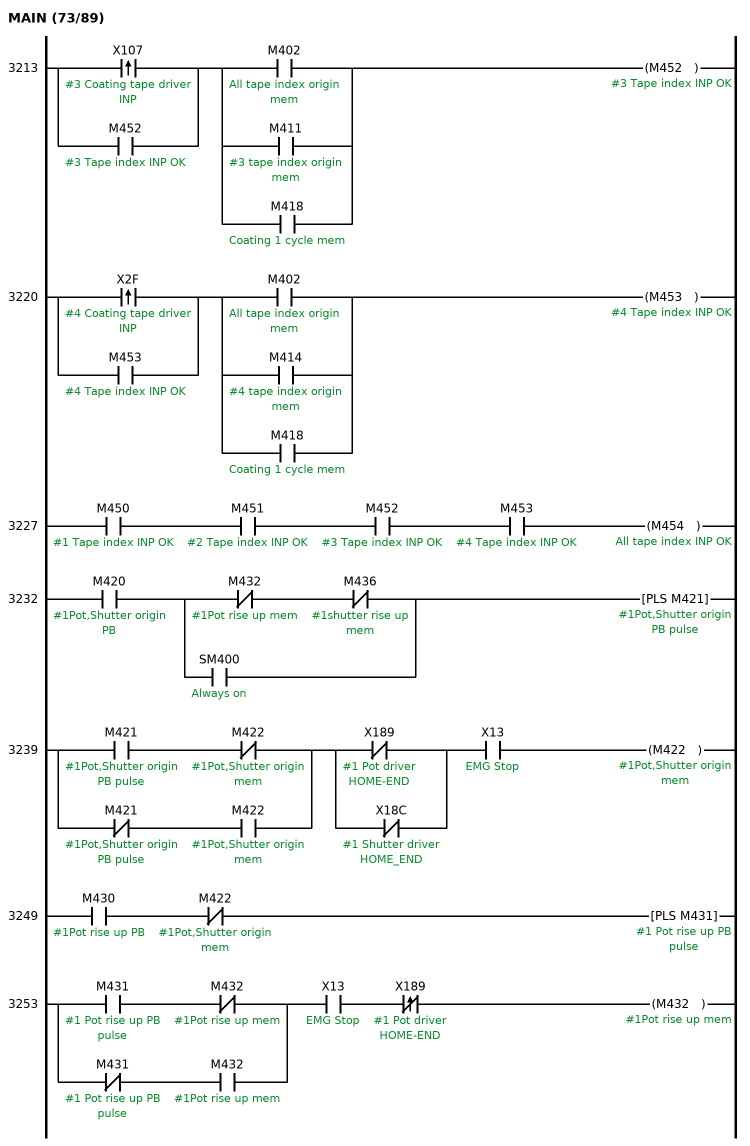
[picture p72: ladder of MAIN, rungs at steps 3213 to 3253]
3213  LDP     X107  ; #3 Coating tape driver INP
      OR      M452  ; #3 Tape index INP OK
      LD      M402  ; All tape index origin mem
      OR      M411  ; #3 tape index origin mem
      OR      M418  ; Coating 1 cycle mem
      ANB
      OUT     M452  ; #3 Tape index INP OK
3220  LDP     X2F  ; #4 Coating tape driver INP
      OR      M453  ; #4 Tape index INP OK
      LD      M402  ; All tape index origin mem
      OR      M414  ; #4 tape index origin mem
      OR      M418  ; Coating 1 cycle mem
      ANB
      OUT     M453  ; #4 Tape index INP OK
3227  LD      M450  ; #1 Tape index INP OK
      AND     M451  ; #2 Tape index INP OK
      AND     M452  ; #3 Tape index INP OK
      AND     M453  ; #4 Tape index INP OK
      OUT     M454  ; All tape index INP OK
3232  LD      M420  ; #1Pot,Shutter origin PB
      LDI     M432  ; #1Pot rise up mem
      ANI     M436  ; #1shutter rise up mem
      OR      SM400  ; Always on
      ANB
      PLS     M421  ; #1Pot,Shutter origin PB pulse
3239  LD      M421  ; #1Pot,Shutter origin PB pulse
      ANI     M422  ; #1Pot,Shutter origin mem
      LDI     M421  ; #1Pot,Shutter origin PB pulse
      AND     M422  ; #1Pot,Shutter origin mem
      ORB
      LDI     X189  ; #1 Pot driver HOME-END
      ORI     X18C  ; #1 Shutter driver HOME_END
      ANB
      AND     X13  ; EMG Stop
      OUT     M422  ; #1Pot,Shutter origin mem
3249  LD      M430  ; #1Pot rise up PB
      ANI     M422  ; #1Pot,Shutter origin mem
      PLS     M431  ; #1 Pot rise up PB pulse
3253  LD      M431  ; #1 Pot rise up PB pulse
      ANI     M432  ; #1Pot rise up mem
      LDI     M431  ; #1 Pot rise up PB pulse
      AND     M432  ; #1Pot rise up mem
      ORB
      AND     X13  ; EMG Stop
      ANDPI   X189  ; #1 Pot driver HOME-END
      OUT     M432  ; #1Pot rise up mem
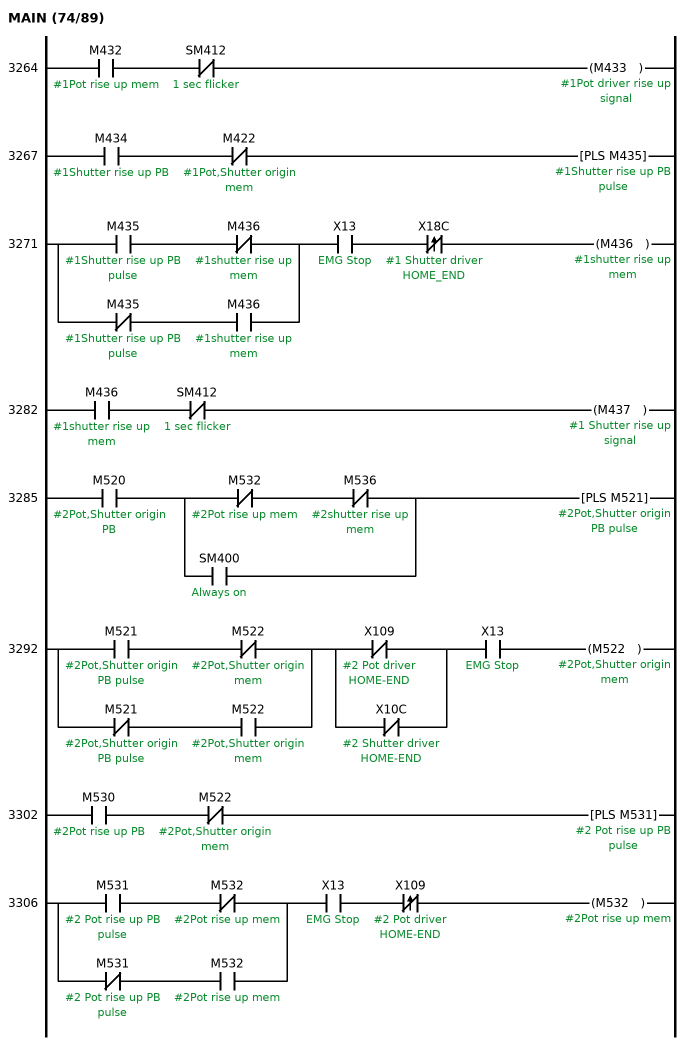
3264  LD      M432  ; #1Pot rise up mem
      ANI     SM412  ; 1 sec flicker
      OUT     M433  ; #1Pot driver rise up signal
3267  LD      M434  ; #1Shutter rise up PB
      ANI     M422  ; #1Pot,Shutter origin mem
      PLS     M435  ; #1Shutter rise up PB pulse
3271  LD      M435  ; #1Shutter rise up PB pulse
      ANI     M436  ; #1shutter rise up mem
      LDI     M435  ; #1Shutter rise up PB pulse
      AND     M436  ; #1shutter rise up mem
      ORB
      AND     X13  ; EMG Stop
      ANDPI   X18C  ; #1 Shutter driver HOME_END
      OUT     M436  ; #1shutter rise up mem
3282  LD      M436  ; #1shutter rise up mem
      ANI     SM412  ; 1 sec flicker
      OUT     M437  ; #1 Shutter rise up signal
3285  LD      M520  ; #2Pot,Shutter origin PB
      LDI     M532  ; #2Pot rise up mem
      ANI     M536  ; #2shutter rise up mem
      OR      SM400  ; Always on
      ANB
      PLS     M521  ; #2Pot,Shutter origin PB pulse
3292  LD      M521  ; #2Pot,Shutter origin PB pulse
      ANI     M522  ; #2Pot,Shutter origin mem
      LDI     M521  ; #2Pot,Shutter origin PB pulse
      AND     M522  ; #2Pot,Shutter origin mem
      ORB
      LDI     X109  ; #2 Pot driver HOME-END
      ORI     X10C  ; #2 Shutter driver HOME-END
      ANB
      AND     X13  ; EMG Stop
      OUT     M522  ; #2Pot,Shutter origin mem
3302  LD      M530  ; #2Pot rise up PB
      ANI     M522  ; #2Pot,Shutter origin mem
      PLS     M531  ; #2 Pot rise up PB pulse
3306  LD      M531  ; #2 Pot rise up PB pulse
      ANI     M532  ; #2Pot rise up mem
      LDI     M531  ; #2 Pot rise up PB pulse
      AND     M532  ; #2Pot rise up mem
      ORB
      AND     X13  ; EMG Stop
      ANDPI   X109  ; #2 Pot driver HOME-END
      OUT     M532  ; #2Pot rise up mem
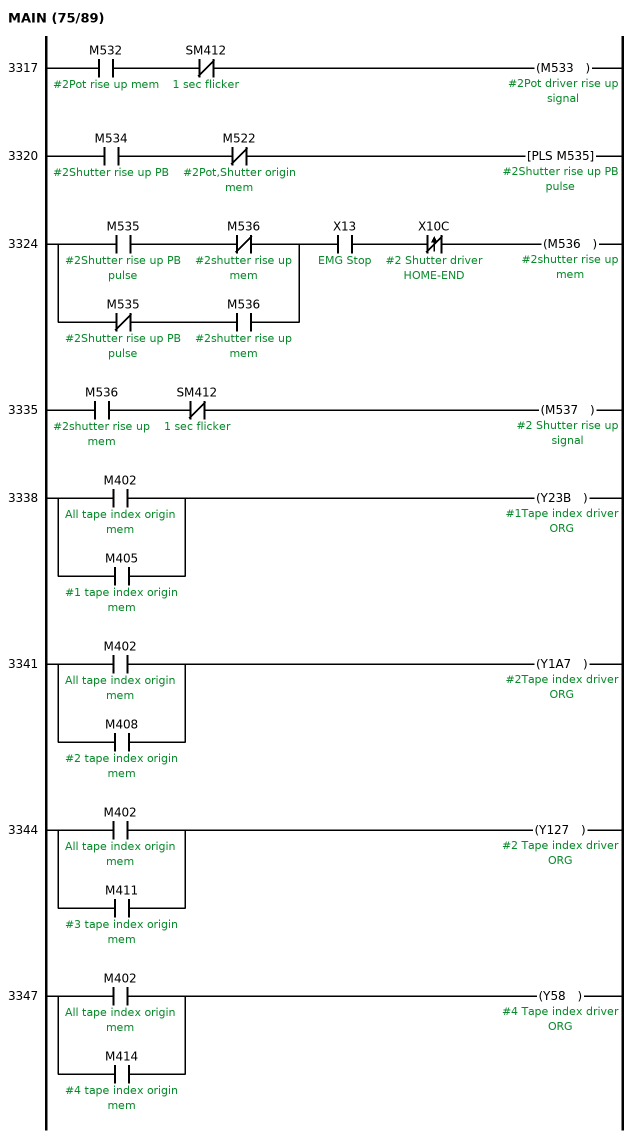
3317  LD      M532  ; #2Pot rise up mem
      ANI     SM412  ; 1 sec flicker
      OUT     M533  ; #2Pot driver rise up signal
3320  LD      M534  ; #2Shutter rise up PB
      ANI     M522  ; #2Pot,Shutter origin mem
      PLS     M535  ; #2Shutter rise up PB pulse
3324  LD      M535  ; #2Shutter rise up PB pulse
      ANI     M536  ; #2shutter rise up mem
      LDI     M535  ; #2Shutter rise up PB pulse
      AND     M536  ; #2shutter rise up mem
      ORB
      AND     X13  ; EMG Stop
      ANDPI   X10C  ; #2 Shutter driver HOME-END
      OUT     M536  ; #2shutter rise up mem
3335  LD      M536  ; #2shutter rise up mem
      ANI     SM412  ; 1 sec flicker
      OUT     M537  ; #2 Shutter rise up signal
3338  LD      M402  ; All tape index origin mem
      OR      M405  ; #1 tape index origin mem
      OUT     Y23B  ; #1Tape index driver ORG
3341  LD      M402  ; All tape index origin mem
      OR      M408  ; #2 tape index origin mem
      OUT     Y1A7  ; #2Tape index driver ORG
3344  LD      M402  ; All tape index origin mem
      OR      M411  ; #3 tape index origin mem
      OUT     Y127  ; #2 Tape index driver ORG
3347  LD      M402  ; All tape index origin mem
      OR      M414  ; #4 tape index origin mem
      OUT     Y58  ; #4 Tape index driver ORG
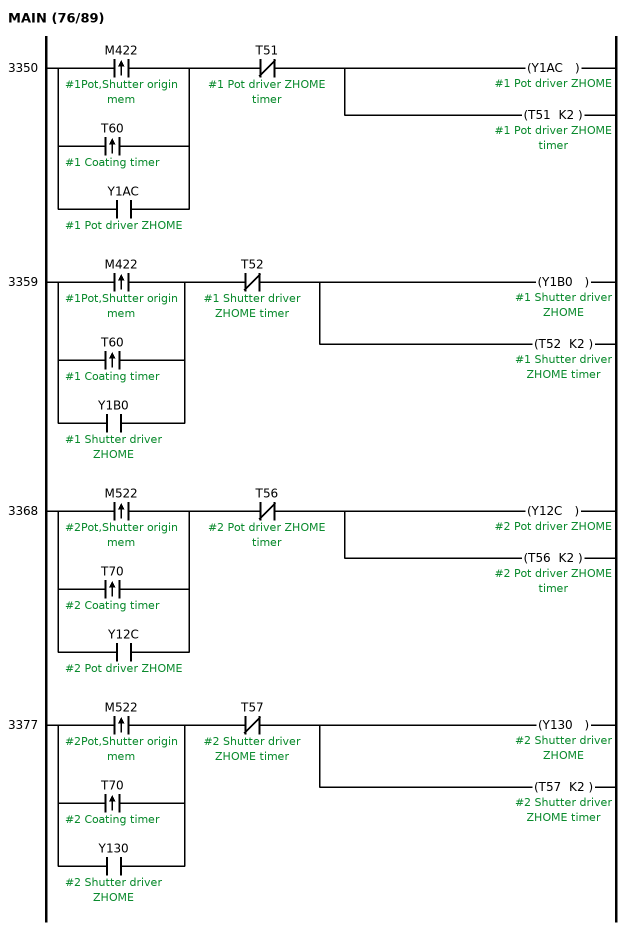
3350  LDP     M422  ; #1Pot,Shutter origin mem
      ORP     T60  ; #1 Coating timer
      OR      Y1AC  ; #1 Pot driver ZHOME
      ANI     T51  ; #1 Pot driver ZHOME timer
      OUT     Y1AC  ; #1 Pot driver ZHOME
      OUT     T51 K2  ; #1 Pot driver ZHOME timer
3359  LDP     M422  ; #1Pot,Shutter origin mem
      ORP     T60  ; #1 Coating timer
      OR      Y1B0  ; #1 Shutter driver ZHOME
      ANI     T52  ; #1 Shutter driver ZHOME timer
      OUT     Y1B0  ; #1 Shutter driver ZHOME
      OUT     T52 K2  ; #1 Shutter driver ZHOME timer
3368  LDP     M522  ; #2Pot,Shutter origin mem
      ORP     T70  ; #2 Coating timer
      OR      Y12C  ; #2 Pot driver ZHOME
      ANI     T56  ; #2 Pot driver ZHOME timer
      OUT     Y12C  ; #2 Pot driver ZHOME
      OUT     T56 K2  ; #2 Pot driver ZHOME timer
3377  LDP     M522  ; #2Pot,Shutter origin mem
      ORP     T70  ; #2 Coating timer
      OR      Y130  ; #2 Shutter driver ZHOME
      ANI     T57  ; #2 Shutter driver ZHOME timer
      OUT     Y130  ; #2 Shutter driver ZHOME
      OUT     T57 K2  ; #2 Shutter driver ZHOME timer
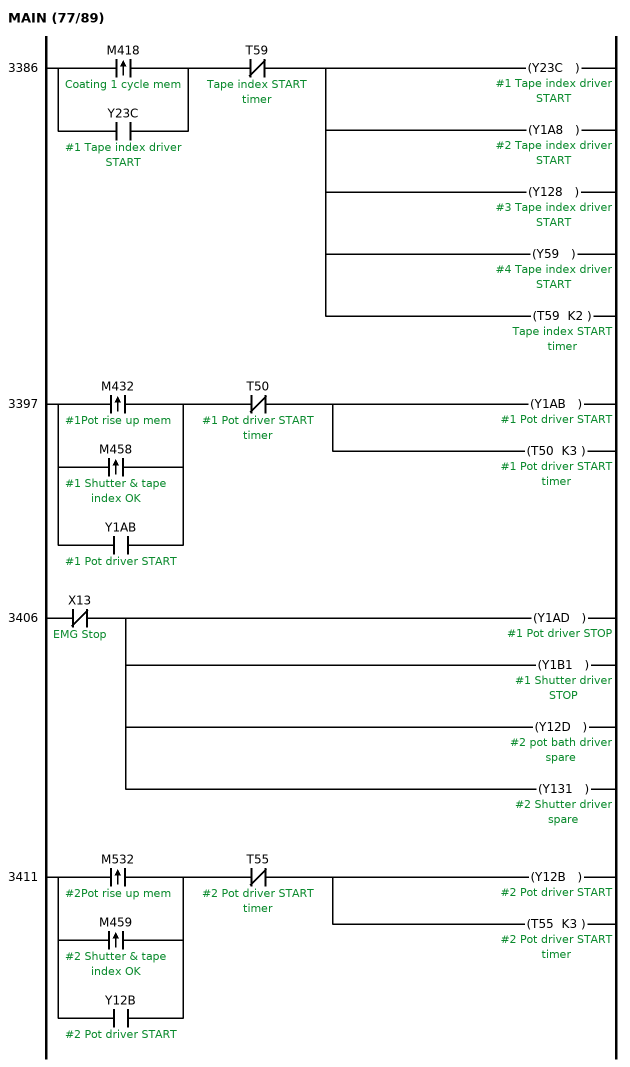
3386  LDP     M418  ; Coating 1 cycle mem
      OR      Y23C  ; #1 Tape index driver START
      ANI     T59  ; Tape index START timer
      OUT     Y23C  ; #1 Tape index driver START
      OUT     Y1A8  ; #2 Tape index driver START
      OUT     Y128  ; #3 Tape index driver START
      OUT     Y59  ; #4 Tape index driver START
      OUT     T59 K2  ; Tape index START timer
3397  LDP     M432  ; #1Pot rise up mem
      ORP     M458  ; #1 Shutter & tape index OK
      OR      Y1AB  ; #1 Pot driver START
      ANI     T50  ; #1 Pot driver START timer
      OUT     Y1AB  ; #1 Pot driver START
      OUT     T50 K3  ; #1 Pot driver START timer
3406  LDI     X13  ; EMG Stop
      OUT     Y1AD  ; #1 Pot driver STOP
      OUT     Y1B1  ; #1 Shutter driver STOP
      OUT     Y12D  ; #2 pot bath driver spare
      OUT     Y131  ; #2 Shutter driver spare
3411  LDP     M532  ; #2Pot rise up mem
      ORP     M459  ; #2 Shutter & tape index OK
      OR      Y12B  ; #2 Pot driver START
      ANI     T55  ; #2 Pot driver START timer
      OUT     Y12B  ; #2 Pot driver START
      OUT     T55 K3  ; #2 Pot driver START timer
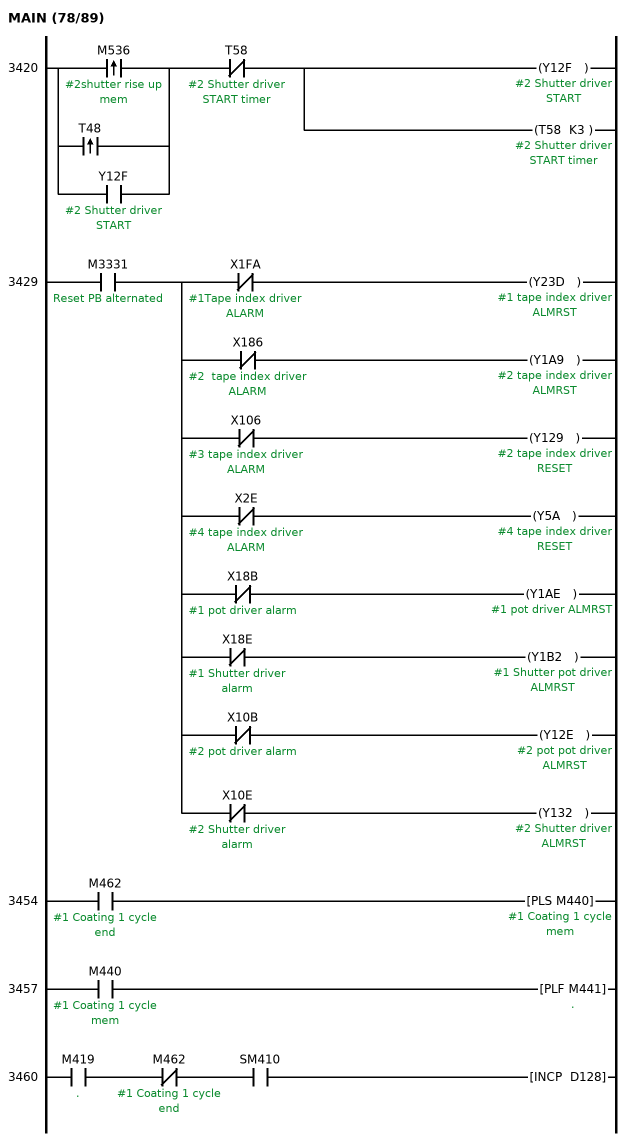
3420  LDP     M536  ; #2shutter rise up mem
      ORP     T48
      OR      Y12F  ; #2 Shutter driver START
      ANI     T58  ; #2 Shutter driver START timer
      OUT     Y12F  ; #2 Shutter driver START
      OUT     T58 K3  ; #2 Shutter driver START timer
3429  LD      M3331  ; Reset PB alternated
      MPS
      ANI     X1FA  ; #1Tape index driver ALARM
      OUT     Y23D  ; #1 tape index driver ALMRST
      MRD
      ANI     X186  ; #2  tape index driver ALARM
      OUT     Y1A9  ; #2 tape index driver ALMRST
      MRD
      ANI     X106  ; #3 tape index driver ALARM
      OUT     Y129  ; #2 tape index driver RESET
      MRD
      ANI     X2E  ; #4 tape index driver ALARM
      OUT     Y5A  ; #4 tape index driver RESET
      MRD
      ANI     X18B  ; #1 pot driver alarm
      OUT     Y1AE  ; #1 pot driver ALMRST
      MRD
      ANI     X18E  ; #1 Shutter driver alarm
      OUT     Y1B2  ; #1 Shutter pot driver ALMRST
      MRD
      ANI     X10B  ; #2 pot driver alarm
      OUT     Y12E  ; #2 pot pot driver ALMRST
      MPP
      ANI     X10E  ; #2 Shutter driver alarm
      OUT     Y132  ; #2 Shutter driver ALMRST
3454  LD      M462  ; #1 Coating 1 cycle end
      PLS     M440  ; #1 Coating 1 cycle mem
3457  LD      M440  ; #1 Coating 1 cycle mem
      PLF     M441  ; .
3460  LD      M419  ; .
      ANI     M462  ; #1 Coating 1 cycle end
      AND     SM410
      INCP    D128
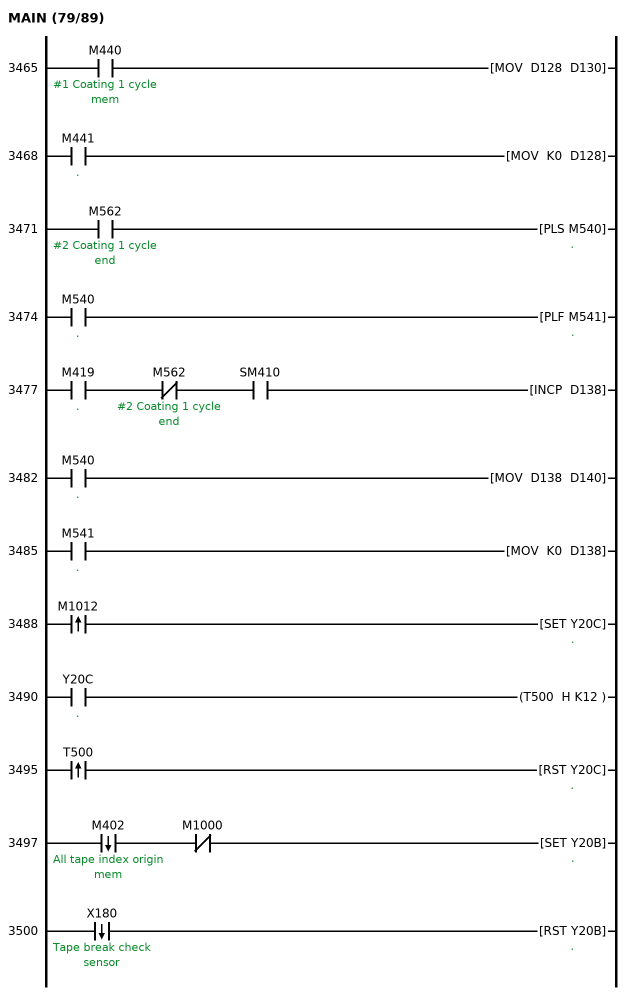
3465  LD      M440  ; #1 Coating 1 cycle mem
      MOV     D128 D130
3468  LD      M441  ; .
      MOV     K0 D128
3471  LD      M562  ; #2 Coating 1 cycle end
      PLS     M540  ; .
3474  LD      M540  ; .
      PLF     M541  ; .
3477  LD      M419  ; .
      ANI     M562  ; #2 Coating 1 cycle end
      AND     SM410
      INCP    D138
3482  LD      M540  ; .
      MOV     D138 D140
3485  LD      M541  ; .
      MOV     K0 D138
3488  LDP     M1012
      SET     Y20C  ; .
3490  LD      Y20C  ; .
      OUTH    T500 K12
3495  LDP     T500
      RST     Y20C  ; .
3497  LDF     M402  ; All tape index origin mem
      ANI     M1000
      SET     Y20B  ; .
3500  LDF     X180  ; Tape break check sensor
      RST     Y20B  ; .
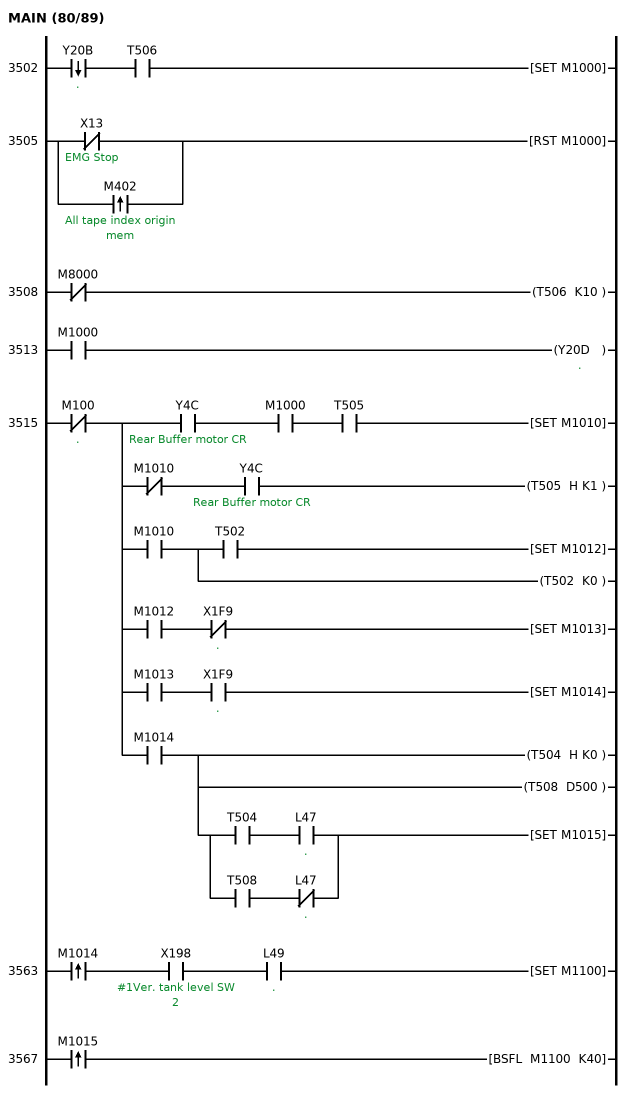
3502  LDF     Y20B  ; .
      AND     T506
      SET     M1000
3505  LDI     X13  ; EMG Stop
      ORP     M402  ; All tape index origin mem
      RST     M1000
3508  LDI     M8000
      OUT     T506 K10
3513  LD      M1000
      OUT     Y20D  ; .
3515  LDI     M100  ; .
      MPS
      AND     Y4C  ; Rear Buffer motor CR
      AND     M1000
      AND     T505
      SET     M1010
      MRD
      ANI     M1010
      AND     Y4C  ; Rear Buffer motor CR
      OUTH    T505 K1
      MRD
      AND     M1010
      MPS
      AND     T502
      SET     M1012
      MPP
      OUT     T502 K0
      MRD
      AND     M1012
      ANI     X1F9  ; .
      SET     M1013
      MRD
      AND     M1013
      AND     X1F9  ; .
      SET     M1014
      MPP
      AND     M1014
      OUTH    T504 K0
      OUT     T508 D500
      LD      T504
      AND     L47  ; .
      LD      T508
      ANI     L47  ; .
      ORB
      ANB
      SET     M1015
3563  LDP     M1014
      AND     X198  ; #1Ver. tank level SW 2
      AND     L49  ; .
      SET     M1100
3567  LDP     M1015
      BSFL    M1100 K40
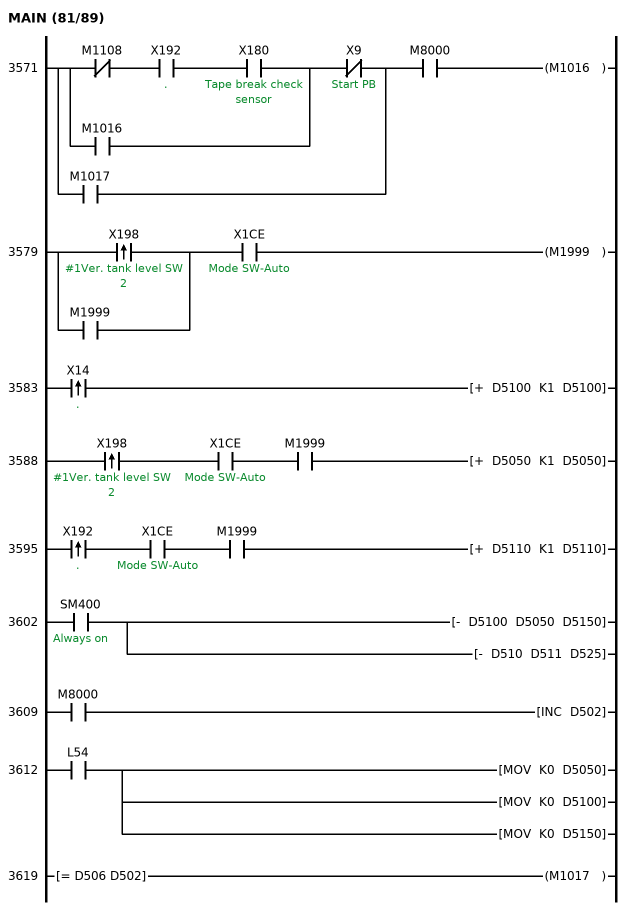
3571  LDI     M1108
      AND     X192  ; .
      AND     X180  ; Tape break check sensor
      OR      M1016
      ANI     X9  ; Start PB
      OR      M1017
      AND     M8000
      OUT     M1016
3579  LDP     X198  ; #1Ver. tank level SW 2
      OR      M1999
      AND     X1CE  ; Mode SW-Auto
      OUT     M1999
3583  LDP     X14  ; .
      +       D5100 K1 D5100
3588  LDP     X198  ; #1Ver. tank level SW 2
      AND     X1CE  ; Mode SW-Auto
      AND     M1999
      +       D5050 K1 D5050
3595  LDP     X192  ; .
      AND     X1CE  ; Mode SW-Auto
      AND     M1999
      +       D5110 K1 D5110
3602  LD      SM400  ; Always on
      -       D5100 D5050 D5150
      -       D510 D511 D525
3609  LD      M8000
      INC     D502
3612  LD      L54
      MOV     K0 D5050
      MOV     K0 D5100
      MOV     K0 D5150
3619  LD=     D506 D502
      OUT     M1017
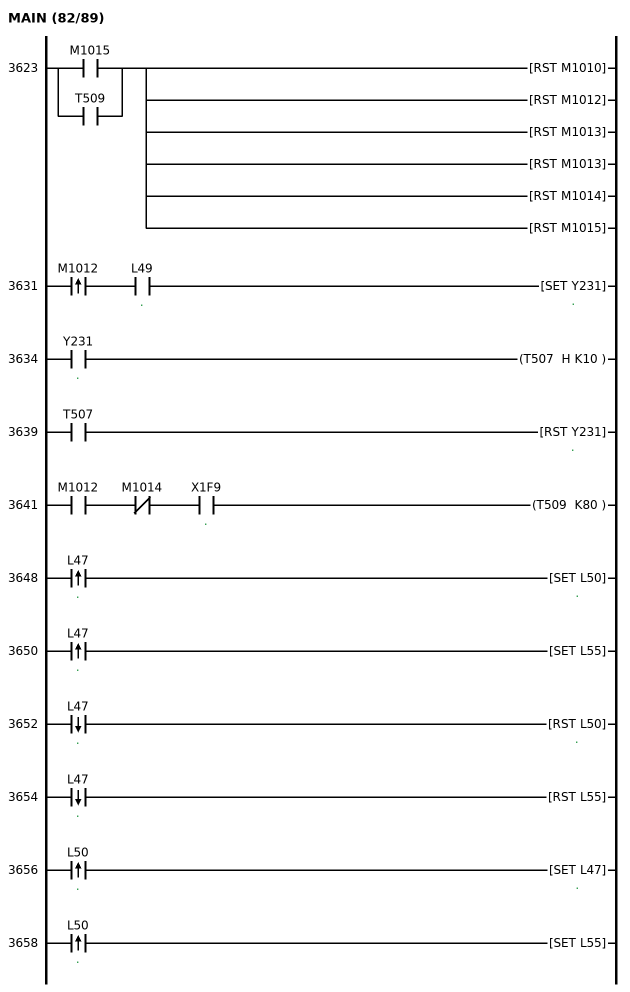
3623  LD      M1015
      OR      T509
      RST     M1010
      RST     M1012
      RST     M1013
      RST     M1013
      RST     M1014
      RST     M1015
3631  LDP     M1012
      AND     L49  ; .
      SET     Y231  ; .
3634  LD      Y231  ; .
      OUTH    T507 K10
3639  LD      T507
      RST     Y231  ; .
3641  LD      M1012
      ANI     M1014
      AND     X1F9  ; .
      OUT     T509 K80
3648  LDP     L47  ; .
      SET     L50  ; .
3650  LDP     L47  ; .
      SET     L55
3652  LDF     L47  ; .
      RST     L50  ; .
3654  LDF     L47  ; .
      RST     L55
3656  LDP     L50  ; .
      SET     L47  ; .
3658  LDP     L50  ; .
      SET     L55
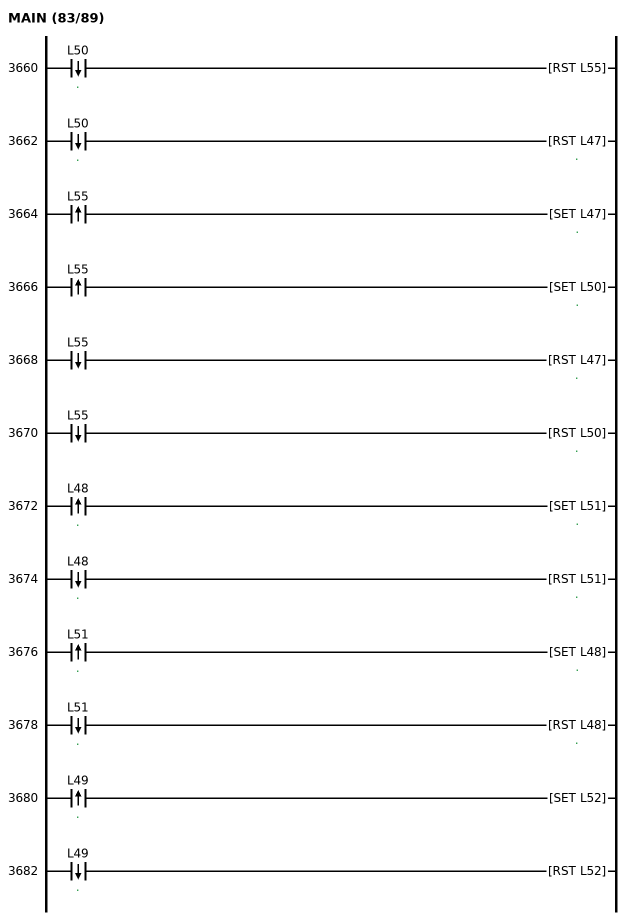
3660  LDF     L50  ; .
      RST     L55
3662  LDF     L50  ; .
      RST     L47  ; .
3664  LDP     L55
      SET     L47  ; .
3666  LDP     L55
      SET     L50  ; .
3668  LDF     L55
      RST     L47  ; .
3670  LDF     L55
      RST     L50  ; .
3672  LDP     L48  ; .
      SET     L51  ; .
3674  LDF     L48  ; .
      RST     L51  ; .
3676  LDP     L51  ; .
      SET     L48  ; .
3678  LDF     L51  ; .
      RST     L48  ; .
3680  LDP     L49  ; .
      SET     L52
3682  LDF     L49  ; .
      RST     L52
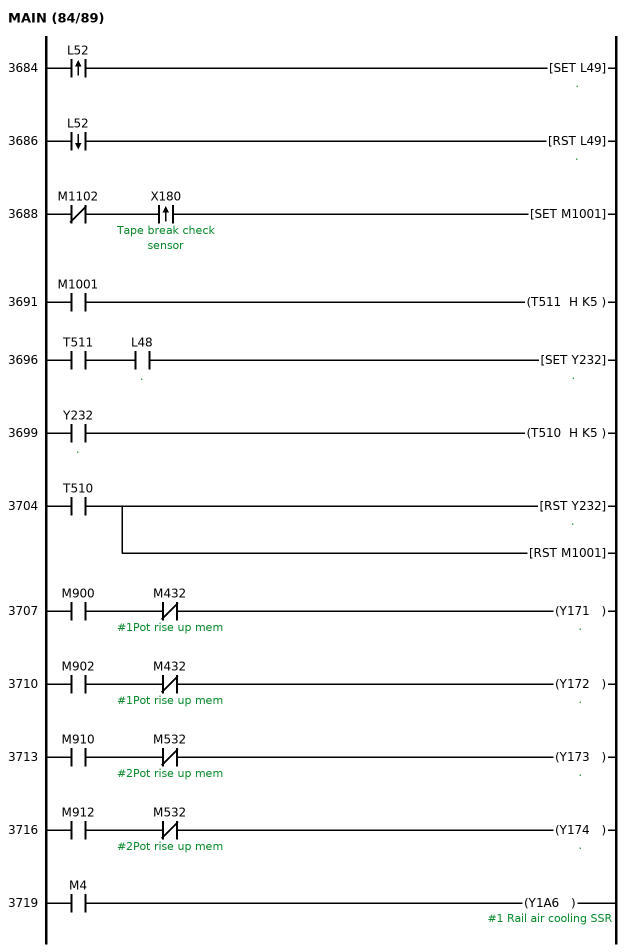
3684  LDP     L52
      SET     L49  ; .
3686  LDF     L52
      RST     L49  ; .
3688  LDI     M1102
      ANDP    X180  ; Tape break check sensor
      SET     M1001
3691  LD      M1001
      OUTH    T511 K5
3696  LD      T511
      AND     L48  ; .
      SET     Y232  ; .
3699  LD      Y232  ; .
      OUTH    T510 K5
3704  LD      T510
      RST     Y232  ; .
      RST     M1001
3707  LD      M900
      ANI     M432  ; #1Pot rise up mem
      OUT     Y171  ; .
3710  LD      M902
      ANI     M432  ; #1Pot rise up mem
      OUT     Y172  ; .
3713  LD      M910
      ANI     M532  ; #2Pot rise up mem
      OUT     Y173  ; .
3716  LD      M912
      ANI     M532  ; #2Pot rise up mem
      OUT     Y174  ; .
3719  LD      M4
      OUT     Y1A6  ; #1 Rail air cooling SSR
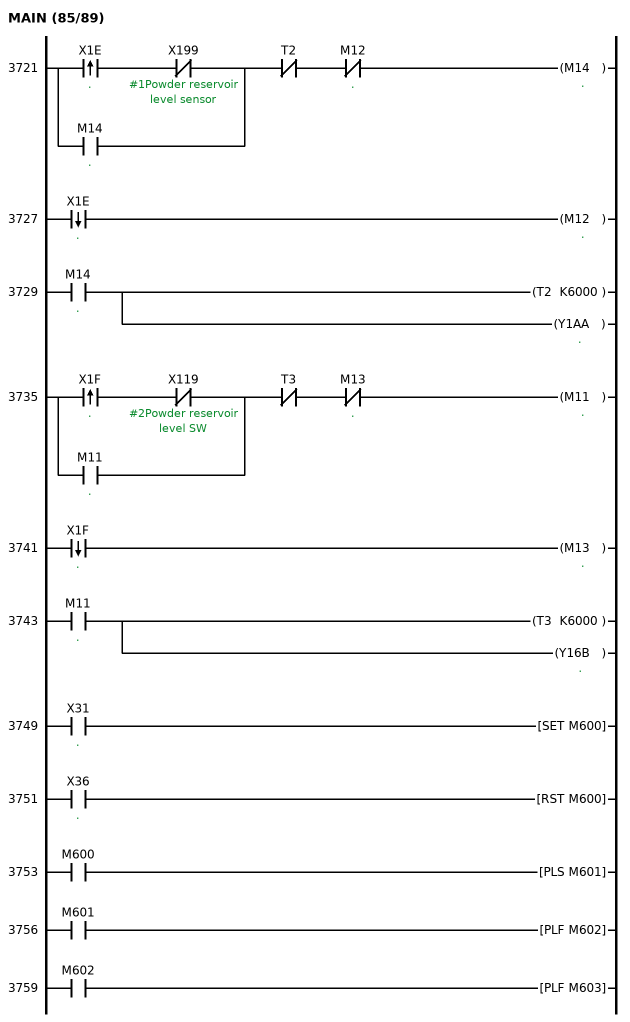
3721  LDP     X1E  ; .
      ANI     X199  ; #1Powder reservoir level sensor
      OR      M14  ; .
      ANI     T2
      ANI     M12  ; .
      OUT     M14  ; .
3727  LDF     X1E  ; .
      OUT     M12  ; .
3729  LD      M14  ; .
      OUT     T2 K6000
      OUT     Y1AA  ; .
3735  LDP     X1F  ; .
      ANI     X119  ; #2Powder reservoir level SW
      OR      M11  ; .
      ANI     T3
      ANI     M13  ; .
      OUT     M11  ; .
3741  LDF     X1F  ; .
      OUT     M13  ; .
3743  LD      M11  ; .
      OUT     T3 K6000
      OUT     Y16B  ; .
3749  LD      X31  ; .
      SET     M600
3751  LD      X36  ; .
      RST     M600
3753  LD      M600
      PLS     M601
3756  LD      M601
      PLF     M602
3759  LD      M602
      PLF     M603
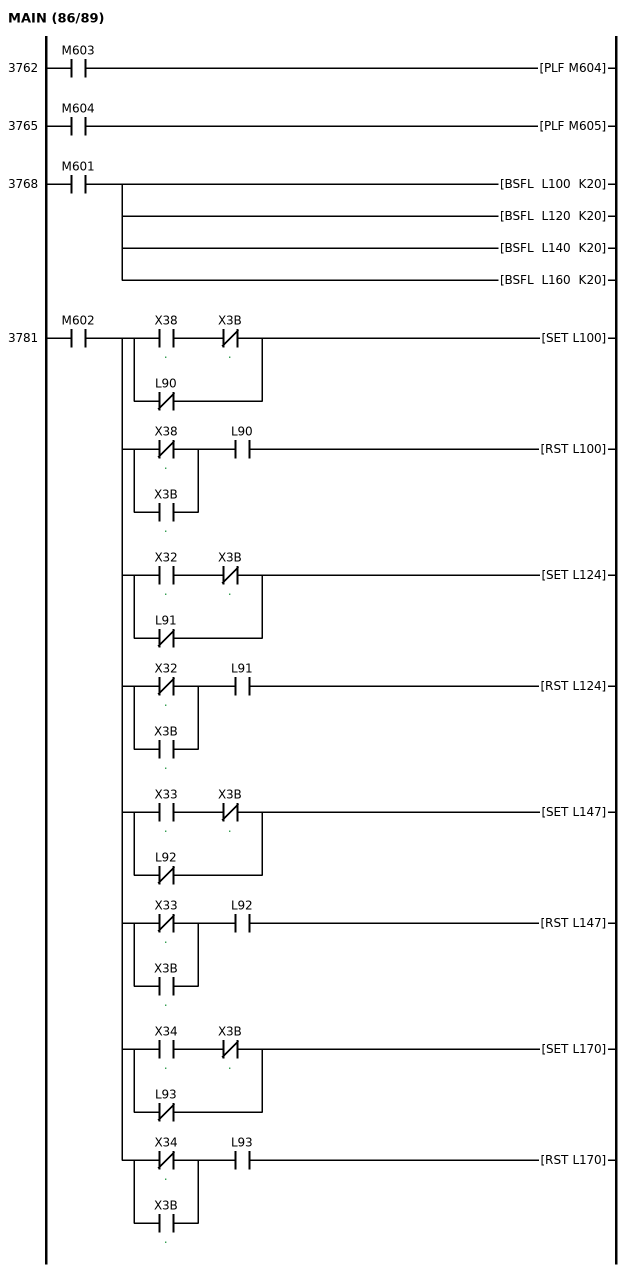
3762  LD      M603
      PLF     M604
3765  LD      M604
      PLF     M605
3768  LD      M601
      BSFL    L100 K20
      BSFL    L120 K20
      BSFL    L140 K20
      BSFL    L160 K20
3781  LD      M602
      MPS
      LD      X38  ; .
      ANI     X3B  ; .
      ORI     L90
      ANB
      SET     L100
      MRD
      LDI     X38  ; .
      OR      X3B  ; .
      ANB
      AND     L90
      RST     L100
      MRD
      LD      X32  ; .
      ANI     X3B  ; .
      ORI     L91
      ANB
      SET     L124
      MRD
      LDI     X32  ; .
      OR      X3B  ; .
      ANB
      AND     L91
      RST     L124
      MRD
      LD      X33  ; .
      ANI     X3B  ; .
      ORI     L92
      ANB
      SET     L147
      MRD
      LDI     X33  ; .
      OR      X3B  ; .
      ANB
      AND     L92
      RST     L147
      MRD
      LD      X34  ; .
      ANI     X3B  ; .
      ORI     L93
      ANB
      SET     L170
      MPP
      LDI     X34  ; .
      OR      X3B  ; .
      ANB
      AND     L93
      RST     L170
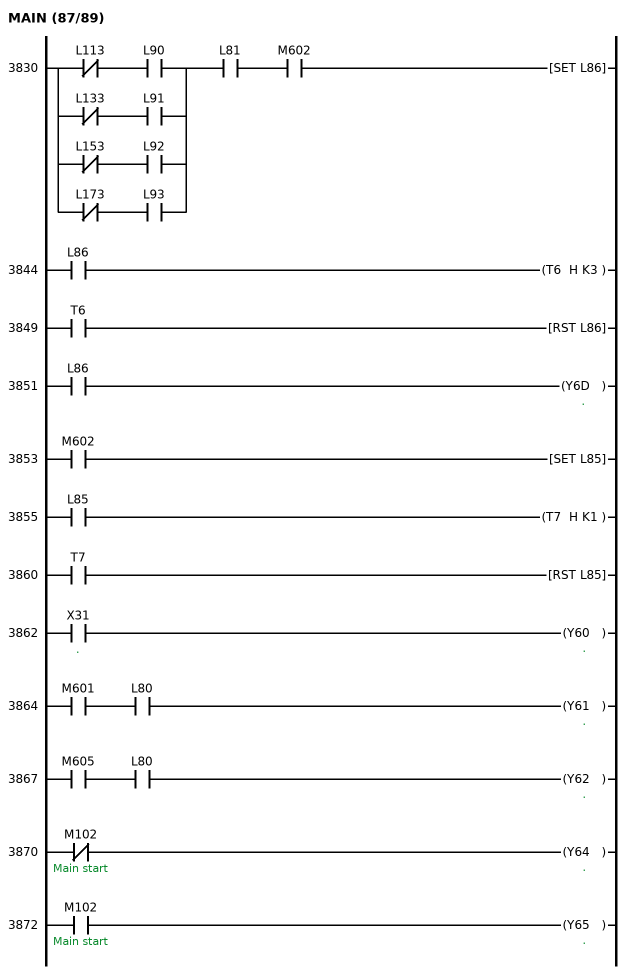
3830  LDI     L113
      AND     L90
      LDI     L133
      AND     L91
      ORB
      LDI     L153
      AND     L92
      ORB
      LDI     L173
      AND     L93
      ORB
      AND     L81
      AND     M602
      SET     L86
3844  LD      L86
      OUTH    T6 K3
3849  LD      T6
      RST     L86
3851  LD      L86
      OUT     Y6D  ; .
3853  LD      M602
      SET     L85
3855  LD      L85
      OUTH    T7 K1
3860  LD      T7
      RST     L85
3862  LD      X31  ; .
      OUT     Y60  ; .
3864  LD      M601
      AND     L80
      OUT     Y61  ; .
3867  LD      M605
      AND     L80
      OUT     Y62  ; .
3870  LDI     M102  ; Main start
      OUT     Y64  ; .
3872  LD      M102  ; Main start
      OUT     Y65  ; .
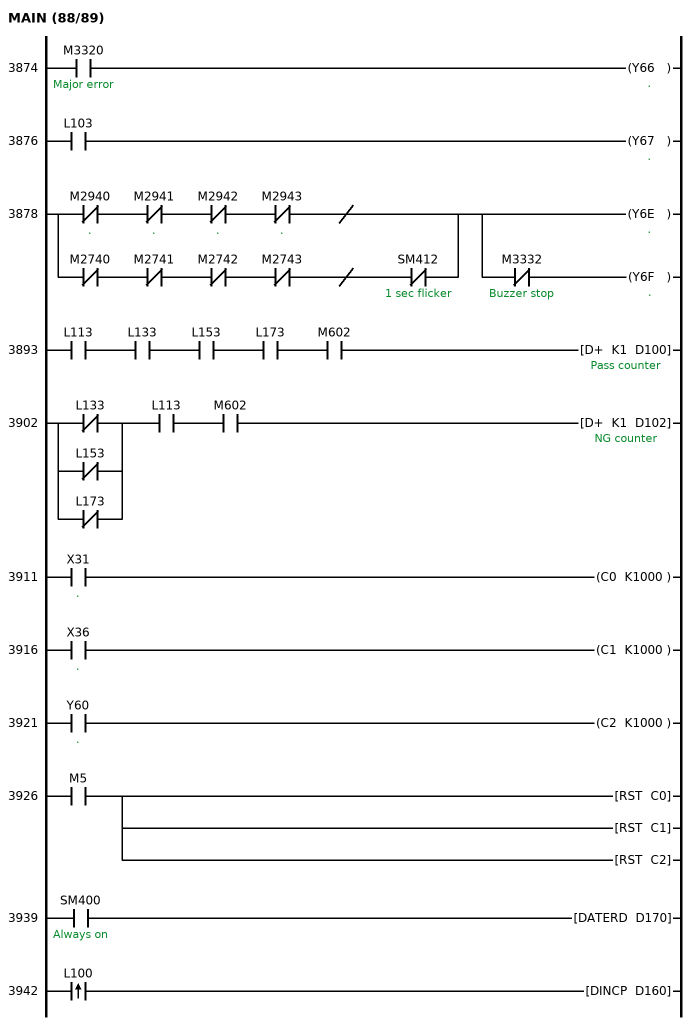
3874  LD      M3320  ; Major error
      OUT     Y66  ; .
3876  LD      L103
      OUT     Y67  ; .
3878  LDI     M2940  ; .
      ANI     M2941  ; .
      ANI     M2942  ; .
      ANI     M2943  ; .
      INV
      LDI     M2740
      ANI     M2741
      ANI     M2742
      ANI     M2743
      INV
      ANI     SM412  ; 1 sec flicker
      ORB
      OUT     Y6E  ; .
      ANI     M3332  ; Buzzer stop
      OUT     Y6F  ; .
3893  LD      L113
      AND     L133
      AND     L153
      AND     L173
      AND     M602
      D+      K1 D100
3902  LDI     L133
      ORI     L153
      ORI     L173
      AND     L113
      AND     M602
      D+      K1 D102
3911  LD      X31  ; .
      OUT     C0 K1000
3916  LD      X36  ; .
      OUT     C1 K1000
3921  LD      Y60  ; .
      OUT     C2 K1000
3926  LD      M5
      RST     C0
      RST     C1
      RST     C2
3939  LD      SM400  ; Always on
      DATERD  D170
3942  LDP     L100
      DINCP   D160
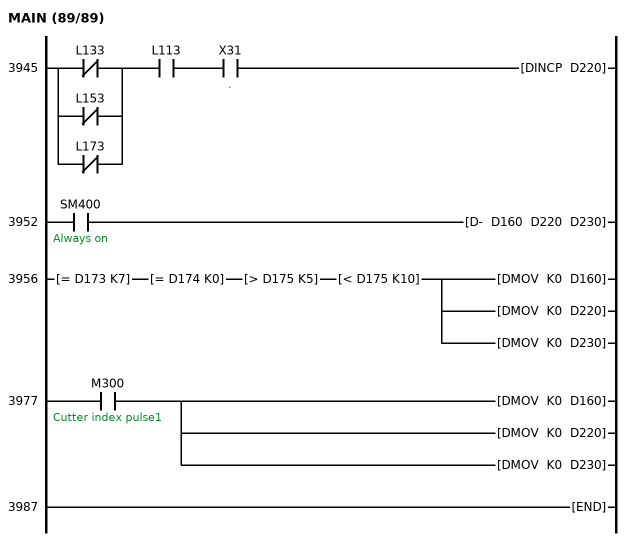
3945  LDI     L133
      ORI     L153
      ORI     L173
      AND     L113
      AND     X31  ; .
      DINCP   D220
3952  LD      SM400  ; Always on
      D-      D160 D220 D230
3956  LD=     D173 K7
      AND=    D174 K0
      AND>    D175 K5
      AND<    D175 K10
      DMOV    K0 D160
      DMOV    K0 D220
      DMOV    K0 D230
3977  LD      M300  ; Cutter index pulse1
      DMOV    K0 D160
      DMOV    K0 D220
      DMOV    K0 D230
3987  END
END_PROGRAM
